// TwinCAT 3 PLC project plc
// ProgramVersion: 3.1.4026.12
// libraries:
//   Tc2_Standard, * (Beckhoff Automation GmbH)
//   Tc2_System, * (Beckhoff Automation GmbH)
//   [Test Framework], * (BA)
// project tree:
//   DUTs/ RecipeData.TcDUT
//   / MAIN.TcPOU, PlcTask.TcTTO
//   POUs/ FB_RecipeValidTest.TcPOU, ValidateRecipe.TcPOU
// real-time tasks:
//   TASK PlcTask: cycle T#10ms, priority 20, ADS port 350

CONFIGURATION plc
    RESOURCE PLC ON TwinCAT3
        TASK PlcTask(INTERVAL := T#10ms, PRIORITY := 20);
        PROGRAM MAIN WITH PlcTask : MAIN;
    END_RESOURCE
END_CONFIGURATION

// ---- DUTs/RecipeData.TcDUT
TYPE RecipeData :
STRUCT
	fTemperature        : REAL;
	nAgitatorSpeed      : DINT;
	nMixTimeSecs        : DINT;	
END_STRUCT
END_TYPE

// ---- MAIN.TcPOU
PROGRAM MAIN
VAR
	fbRecipeTest_Valid              : FB_RecipeValidTest(sTestName:='Recipe Valid') := 
										(bExpected:= TRUE);
	fbRecipeTest_InvalidLoTemp      : FB_RecipeValidTest(sTestName:='Recipe Invalid Lo Temp') := 
										(bExpected:= FALSE, 
										MockRecipe:=(fTemperature:=139.9));
	fbRecipeTest_InvalidHiTemp      : FB_RecipeValidTest(sTestName:='Recipe Invalid Hi Temp') := 
										(bExpected:= FALSE,
										MockRecipe:=(fTemperature:=185.1));
	fbTestRunner                    : FB_TestRunner;
	bInit                           : BOOL;								
END_VAR

// run once
IF NOT bInit THEN
    fbTestRunner.AddTest(fbRecipeTest_Valid);
    fbTestRunner.AddTest(fbRecipeTest_InvalidLoTemp);
    fbTestRunner.AddTest(fbRecipeTest_InvalidHiTemp);
    bInit := TRUE;
END_IF
fbTestRunner.Execute();

END_PROGRAM

// ---- POUs/FB_RecipeValidTest.TcPOU
FUNCTION_BLOCK FB_RecipeValidTest EXTENDS FB_SimpleTest
VAR_INPUT
	bExpected       : BOOL;
	MockRecipe      : RecipeData := (
                        fTemperature:=140.0, 
                        nAgitatorSpeed:=10, 
                        nMixTimeSecs:=300
                    );
END_VAR
VAR_OUTPUT
END_VAR
VAR
END_VAR

METHOD Execute : BOOL
VAR_INPUT
END_VAR
VAR_INST
	bResult		: BOOL;
END_VAR
bResult := ValidateRecipe(MockRecipe);
AssertEquals(bExpected, bResult, 'Recipe validation failed');
Execute := TRUE;
END_METHOD

END_FUNCTION_BLOCK

// ---- POUs/ValidateRecipe.TcPOU
FUNCTION ValidateRecipe : Bool
VAR_INPUT
	Recipe          : REFERENCE TO RecipeData;
END_VAR
VAR
END_VAR

ValidateRecipe :=
    (Recipe.fTemperature >= 140.0 AND Recipe.fTemperature <= 185.0) AND
    (Recipe.nAgitatorSpeed >= 10 AND Recipe.nAgitatorSpeed <= 100) AND
    (Recipe.nMixTimeSecs >= 300 AND Recipe.nMixTimeSecs <= 500);

END_FUNCTION
